FUNCTION_BLOCK CentralServer (* Basic Function Block Type *)
  (* Standard: 61499-2 *)
  (* Version 0.2, 2003-12-04, JHC, Rockwell Automation, Renamed for better indexing. *)
  (* Version 0.1, 2002-11-05, JHC, Rockwell Automation, Corrected missing ST element in Algorithm REQ. *)
  (* Version 0.0, 2000-05-30, JHC, Rockwell Automation *)
  (* Compiler header: package fb.rt.conveyorIEC61499; *)
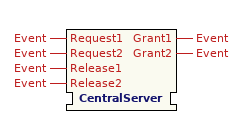
  EVENT_INPUT
    Request1;
    Request2;
    Release1;
    Release2;
  END_EVENT
  EVENT_OUTPUT
    Grant1;
    Grant2;
  END_EVENT
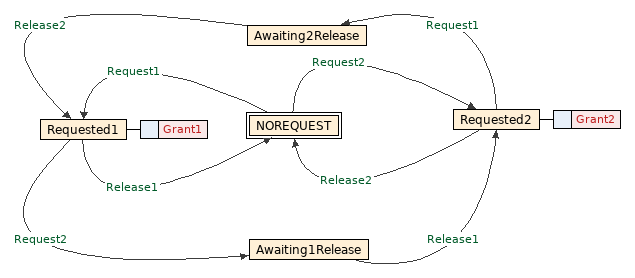
  EC_STATES
    NOREQUEST; (* Initial State *)
    Requested1 : -> Grant1;
    Requested2 : -> Grant2;
    Awaiting1Release;
    Awaiting2Release;
  END_STATES
  EC_TRANSITIONS
    NOREQUEST TO Requested2 := Request2;
    NOREQUEST TO Requested1 := Request1;
    Requested2 TO NOREQUEST := Release2;
    Requested1 TO NOREQUEST := Release1;
    Requested1 TO Awaiting1Release := Request2;
    Awaiting1Release TO Requested2 := Release1;
    Requested2 TO Awaiting2Release := Request1;
    Awaiting2Release TO Requested1 := Release2;
  END_TRANSITIONS
END_FUNCTION_BLOCK
